(* CODESYS project Broadcast.library
   Company: _
   DefaultNamespace: Broadcast
   Title: Broadcast
   Placeholder: _Broadcast
   Author: Krystian Lis et al.
   Description: Sub-pub com.
   Version: 1.0.0

Project tree, tasks and I/O mapping:
  libraries: Debug, * (_); Results, * (_); Strings, * (_); Tags, * (_); Utils, * (_); Tc2_Standard, * (Beckhoff Automation GmbH); Tc2_System, * (Beckhoff Automation GmbH); Domains, * (_); Calls, * (_)
  Broadcast/
    _/
      Helpers/
        function _ArePaired [ST]
        function _Cleanup [ST]
        function _Clear [ST]
        function _Copy [ST]
        function _EmitSignal [ST]
        function _FindBestChunk [ST]
        function _FindChunkAfter [ST]
        function _NewPair [ST]
        function _SoftCompress [ST]
        function _Unpair [ST]
      Structs/
        data type ST_Entry
    Receiver/
      interface I_Receiver: Pair, Unpair
      interface I_ReceiverNode: IsOk, Receive
      function block Receiver [ST]: FB_init, IsOk, Pair, Receive, Tag, Unpair
    Signal/
      function block EmitProxy [ST]: FB_init
      interface I_Emit: Emit, EmitTo, Option, Pair, Unpair
      interface I_Signal: Pair, Unpair
      interface I_SignalNode: count, id, size
      function block Signal [ST]: count, id, size, Emit, EmitTo, FB_init, Option, Pair, Tag, Unpair
    global variables _Channel
    global variables Param
*)

// Broadcast/_/Structs/ST_Entry
TYPE INTERNAL ST_Entry :
STRUCT
	iSignal		: I_SignalNode;
	iReceiver	: I_ReceiverNode;
END_STRUCT
END_TYPE

// Broadcast/_Channel
{attribute 'qualified_only'}
VAR_GLOBAL INTERNAL
	{attribute 'ExpandFully'} 
	// Fixed-size array to store all signal-receiver entries.
	// Index 0 is reserved and not used (signals with id = 0 are unassigned).
	stEntry				: ARRAY[0..Param.nChannelSize] OF ST_Entry;
	
	// Total number of assigned entries in the stEntry array.
	nAssigned			: UDINT;
END_VAR

// Broadcast/Param
{attribute 'qualified_only'}
VAR_GLOBAL CONSTANT
	nChannelSize		: UDINT(1..16#FFFFFFE) := 100;
END_VAR

// Broadcast/_/Helpers/_ArePaired
FUNCTION INTERNAL _ArePaired : BOOL
VAR_INPUT
	iSignal				: I_SignalNode;
    iReceiver			: I_ReceiverNode;
END_VAR
VAR_OUTPUT
	nPos				: UDINT;
END_VAR
VAR
	i					: UDINT;
	_nEnd				: UDINT;
END_VAR

IF iSignal.count = 0 THEN
	_ArePaired := FALSE;
	RETURN;	
END_IF

_nEnd := iSignal.id + iSignal.count - 1;
FOR i := iSignal.id TO _nEnd DO
	IF _Channel.stEntry[i].iReceiver = iReceiver THEN
		_ArePaired := TRUE;
		nPos := i;
		RETURN;
	END_IF
END_FOR

END_FUNCTION

// Broadcast/Signal/I_SignalNode
INTERFACE INTERNAL I_SignalNode EXTENDS Debug.I_Debug

PROPERTY INTERNAL count : UDINT
GET
END_GET
SET
END_SET
END_PROPERTY

PROPERTY INTERNAL id : UDINT
GET
END_GET
SET
END_SET
END_PROPERTY

PROPERTY INTERNAL size : UDINT
GET
END_GET
SET
END_SET
END_PROPERTY

END_INTERFACE

// Broadcast/Receiver/I_ReceiverNode
INTERFACE INTERNAL I_ReceiverNode EXTENDS Debug.I_Debug

PROPERTY INTERNAL IsOk : BOOL
GET
END_GET
END_PROPERTY

METHOD INTERNAL Receive
VAR_INPUT
	iArg			: Calls.I_Arg;
END_VAR
END_METHOD

END_INTERFACE

// Broadcast/_/Helpers/_Cleanup
FUNCTION INTERNAL _Cleanup
VAR
	i					: UDINT;
	_iSignal			: I_SignalNode;
END_VAR

// Loop through stEntry to update signal ids
FOR i := 1 TO Param.nChannelSize DO
	IF _Channel.stEntry[i].iSignal <> 0 AND_THEN _Channel.stEntry[i].iSignal <> _iSignal THEN
			_iSignal := _Channel.stEntry[i].iSignal;
			_iSignal.id := i;
	END_IF
END_FOR

END_FUNCTION

// Broadcast/Signal/Signal
FUNCTION_BLOCK FINAL Signal IMPLEMENTS I_SignalNode, I_Signal, Tags.I_Tagged, I_Emit
VAR
	_tag			: Tags.Tag;
	_nCount			: UDINT;
	_nSize			: UDINT;
	_nId			: UDINT;
END_VAR

PROPERTY INTERNAL count : UDINT
GET
count := _nCount;
END_GET
SET
_nCount := count;
END_SET
END_PROPERTY

PROPERTY INTERNAL id : UDINT
GET
id := _nId;
END_GET
SET
_nId := id;
END_SET
END_PROPERTY

PROPERTY INTERNAL size : UDINT
GET
size := _nSize;
END_GET
SET
_nSize := size;
END_SET
END_PROPERTY

METHOD Emit
VAR_INPUT
	iArg			: Calls.I_Arg := 0;
END_VAR
IF iArg = 0 THEN
	iArg := Calls.Arg.phantom;
END_IF

_EmitSignal(THIS^, iArg);
END_METHOD

METHOD EmitTo : Results.Result
VAR_INPUT
	iReceiver		: I_Receiver;
	iArg			: Calls.I_Arg;
END_VAR
IF iReceiver = 0 THEN
	EmitTo := Results.Err.Itf0;
	RETURN;
END_IF

IF iArg = 0 THEN
	iArg := Calls.Arg.phantom;
END_IF

iReceiver.Receive(iArg);
EmitTo := Results.Ok;
END_METHOD

//FB_Init is always available implicitly and it is used primarily for initialization.
//The return value is not evaluated. For a specific influence, you can also declare the
//methods explicitly and provide additional code there with the standard initialization
//code. You can evaluate the return value.
METHOD FB_Init: BOOL
VAR_INPUT
    bInitRetains: BOOL; // TRUE: the retain variables are initialized (reset warm / reset cold)
    bInCopyCode: BOOL;  // TRUE: the instance will be copied to the copy code afterward (online change)

	iCTable		: Domains.I_MutCTable;
END_VAR
VAR
	_nResult		: Results.Result;
END_VAR
IF iCTable <> 0 THEN
	CASE (_nResult := iCTable.Insert(THIS^)) OF
		Results.Ok:	
			// Do nothing
		Results.Err.ItfEq:
			Debug.DebugMsg(THIS^, 'Alredy exist within iCTable!');
			Debug.DebugMsg(iCTable, '^');
		Results.Err.Ovf:
			Debug.DebugMsg(THIS^, 'iCTable overflow!');
		ELSE
			Debug.DebugMsg(THIS^, Tc2_Standard.CONCAT(TO_STRING(_nResult), ': Unknown error'));
	END_CASE

ELSE
	Debug.DebugMsg(THIS^, 'iCTable = 0!');
END_IF
END_METHOD

METHOD Option : REFERENCE TO Signal
VAR_INPUT
	sOption		: Strings.Str;
END_VAR
Option REF= THIS^;
_tag.Option := sOption;
END_METHOD

METHOD Pair : Results.Result
VAR_INPUT
	iReceiver		: I_Receiver;
END_VAR
IF iReceiver = 0 THEN
	Pair := Results.Err.Itf0;
ELSIF iReceiver.IsOk THEN
	Pair := _NewPair(THIS^, iReceiver);
ELSE
	Pair := Results.Error;
END_IF
END_METHOD

PROPERTY Tag : Tags.I_Tag
GET
Tag := _tag;
END_GET
END_PROPERTY

METHOD Unpair : Results.Result
VAR_INPUT
	iReceiver		: I_Receiver;
END_VAR
IF iReceiver = 0 THEN
	Unpair := Results.Err.Itf0;
ELSIF iReceiver.IsOk THEN
	Unpair := _Unpair(THIS^, iReceiver);
ELSE
	Unpair := Results.Error;
END_IF
END_METHOD

END_FUNCTION_BLOCK

// Broadcast/Signal/I_Signal
INTERFACE I_Signal EXTENDS Debug.I_Debug, Domains.I_Component

METHOD Pair : Results.Result
VAR_INPUT
	iReceiver		: I_Receiver;
END_VAR
END_METHOD

METHOD Unpair : Results.Result
VAR_INPUT
	iReceiver		: I_Receiver;
END_VAR
END_METHOD

END_INTERFACE

// Broadcast/Receiver/I_Receiver
INTERFACE I_Receiver EXTENDS I_ReceiverNode, Domains.I_Component;

METHOD Pair : Results.Result
VAR_INPUT
	iSignal		: I_Signal;
END_VAR
END_METHOD

METHOD Unpair : Results.Result
VAR_INPUT
	iSignal		: I_Signal;
END_VAR
END_METHOD

END_INTERFACE

// Broadcast/Signal/I_Emit
INTERFACE I_Emit

METHOD Emit
VAR_INPUT
	iArg			: Calls.I_Arg;
END_VAR
END_METHOD

METHOD EmitTo : Results.Result
VAR_INPUT
	iReceiver		: I_Receiver;
	iArg			: Calls.I_Arg;
END_VAR
END_METHOD

METHOD Option : REFERENCE TO Signal
VAR_INPUT
	sOption		: Strings.Str;
END_VAR
END_METHOD

METHOD Pair : Results.Result
VAR_INPUT
	iReceiver		: I_Receiver;
END_VAR
END_METHOD

METHOD Unpair : Results.Result
VAR_INPUT
	iReceiver		: I_Receiver;
END_VAR
END_METHOD

END_INTERFACE

// Broadcast/_/Helpers/_EmitSignal
FUNCTION INTERNAL _EmitSignal
VAR_INPUT
	iSignal		: I_SignalNode;
	iArg		: Calls.I_Arg;
END_VAR
VAR
	i			: UDINT;
	nEnd		: UDINT;
END_VAR

IF iSignal.count = 0 THEN
	RETURN;
END_IF

nEnd := iSignal.id + iSignal.count - 1;
FOR i := iSignal.id TO nEnd DO
	_Channel.stEntry[i].iReceiver.Receive(iArg);
END_FOR

END_FUNCTION

// Broadcast/_/Helpers/_NewPair
FUNCTION INTERNAL _NewPair : Results.Result
VAR_INPUT
	iSignal				: I_SignalNode;
	iReceiver			: I_ReceiverNode;
END_VAR
VAR
	_nSignalSize		: UDINT;
	_nSignalCount		: UDINT;
	_nSignalId			: UDINT;
	
	_nNewId				: UDINT;
	_nNewSize			: UDINT;
	_nRequestedSize		: UDINT;
	_nDiff				: UDINT;
	
	_nFree				: UDINT;
	
	_bReallocation		: BOOL;
END_VAR

//If itfs are 0
IF iSignal = 0 OR iReceiver = 0 THEN
	_NewPair := Results.Err.Itf0;
	RETURN;
END_IF	
//If pair already exist
IF _ArePaired(iSignal, iReceiver) THEN
	_NewPair := Results.None;
	RETURN;
END_IF
// First signal ever
IF _Channel.nAssigned = 0 THEN
	_Channel.stEntry[1].iSignal := iSignal;
	_Channel.stEntry[1].iReceiver := iReceiver;
	iSignal.id := 1;
	iSignal.size := 1;
	iSignal.count := 1;
	_Channel.nAssigned := 1;;
	_NewPair := Results.Ok;
	RETURN;	
END_IF

//If signal has enough space
IF (_nSignalCount := iSignal.count) > 0 AND_THEN _nSignalCount < (_nSignalSize := iSignal.size) THEN
	_Channel.stEntry[iSignal.id + _nSignalCount].iSignal := iSignal;
	_Channel.stEntry[iSignal.id + _nSignalCount].iReceiver := iReceiver;
	iSignal.count := _nSignalCount + 1;
	_NewPair := Results.Ok;
	RETURN;
END_IF

IF iSignal.id <> 0 THEN
	//If signal has enough space after
	IF Results.IsOk(_FindChunkAfter(_nSignalSize + (_nSignalId := iSignal.id), 1, nNewSize => _nNewSize)) THEN
		_Channel.stEntry[iSignal.id + _nSignalCount].iSignal := iSignal;
		_Channel.stEntry[iSignal.id + _nSignalCount].iReceiver := iReceiver;
		iSignal.size := _nNewSize + _nSignalSize;
		iSignal.count := _nSignalCount + 1;
		_Channel.nAssigned := _Channel.nAssigned + 1;
		_NewPair := Results.Ok;
		RETURN;
	END_IF
END_IF

// What new size should be
IF (_nFree := Param.nChannelSize - _Channel.nAssigned) >= _nSignalSize + 1 THEN
	_nRequestedSize := _nSignalSize + 1;
ELSE
	_NewPair := Results.Err.Ovf;
	RETURN;
END_IF

_nSignalId := iSignal.id;
IF Results.IsOk(_FindBestChunk(_nSignalId, _nRequestedSize, nNewId => _nNewId, nNewSize => _nNewSize)) THEN
	IF _nSignalId <> 0 THEN
		_Copy(_nSignalId, _nSignalSize, _nNewId);
		_Clear(_nSignalId, _nSignalSize);		
	END_IF		
	_Channel.stEntry[_nNewId + _nSignalCount].iSignal := iSignal;
	_Channel.stEntry[_nNewId + _nSignalCount].iReceiver := iReceiver;
	iSignal.id := _nNewId;
	iSignal.size := _nNewSize;
	iSignal.count := _nSignalCount + 1;
	_Channel.nAssigned := _Channel.nAssigned - _nSignalSize + _nNewSize;
	_NewPair := Results.Ok;	
	RETURN;
END_IF

_SoftCompress();
_Cleanup();


_nSignalId := iSignal.id; // _nSignalId needs to be revalidated.
IF Results.IsOk(_FindBestChunk(_nSignalId, _nRequestedSize, nNewId => _nNewId, nNewSize => _nNewSize)) THEN
	IF _nSignalId <> 0 THEN
		_Copy(_nSignalId, _nSignalSize, _nNewId);
		_Clear(_nSignalId, _nSignalSize);		
	END_IF
	_Channel.stEntry[_nNewId + _nSignalCount].iSignal := iSignal;
	_Channel.stEntry[_nNewId + _nSignalCount].iReceiver := iReceiver;
	iSignal.id := _nNewId;
	iSignal.size := _nNewSize;
	iSignal.count := _nSignalCount + 1;
	_Channel.nAssigned := _Channel.nAssigned - _nSignalSize + _nNewSize;
	_NewPair := Results.Ok;	
	RETURN;
END_IF

_NewPair := Results.Error;

END_FUNCTION

// Broadcast/_/Helpers/_FindChunkAfter
FUNCTION INTERNAL _FindChunkAfter : Results.Result
VAR_INPUT
	nId					: UDINT;
    nRequestedSize     	: UDINT;
END_VAR
VAR_OUTPUT
    nNewSize            : UDINT;
END_VAR
VAR
	i					: UDINT;
END_VAR

// Loop from the starting index to the end of stEntry
FOR i := nId TO Param.nChannelSize DO
	IF nRequestedSize = nNewSize THEN
		EXIT;
	ELSIF _Channel.stEntry[i].iSignal = 0 THEN
		nNewSize := nNewSize + 1;
	ELSE
		EXIT;
	END_IF
END_FOR

// Check if the required size was found
IF nNewSize = nRequestedSize THEN
	_FindChunkAfter := Results.Ok;
ELSE
	_FindChunkAfter := Results.Error;
END_IF

END_FUNCTION

// Broadcast/_/Helpers/_FindBestChunk
FUNCTION INTERNAL _FindBestChunk : Results.Result
VAR_INPUT
	nRequesterId		: UDINT;
    nRequestedSize     	: UDINT;
END_VAR
VAR_OUTPUT
    nNewId             	: UDINT;
    nNewSize            : UDINT;
END_VAR
VAR
	i					: UDINT;
	j					: UDINT;
END_VAR

// Loop through stEntry to find the best chunk
FOR i := 1 TO Param.nChannelSize DO
	IF _Channel.stEntry[i].iSignal <> 0 AND_THEN _Channel.stEntry[i].iSignal.id <> nRequesterId THEN
		// Skip over occupied blocks
		i := _Channel.stEntry[i].iSignal.id + _Channel.stEntry[i].iSignal.size - 1;
	ELSE
		// Start of a free chunk and measure its size
		FOR j := 0 TO Param.nChannelSize DO
			IF _Channel.stEntry[i + j].iSignal <> 0 AND_THEN _Channel.stEntry[i].iSignal.id <> nRequesterId THEN
				EXIT;
			ELSIF Param.nChannelSize <= i + j THEN
				EXIT;
			END_IF			
		END_FOR
		
		// If the chunk is smaller but still fits assign a new best fit
		IF nNewSize = 0 THEN
			nNewId := i;
			nNewSize := j + 1;
		ELSIF  nRequestedSize <= j + 1 AND_THEN nNewSize > j + 1 THEN
			nNewId := i;
			nNewSize := nRequestedSize;
		END_IF
		
		IF _Channel.stEntry[i + j].iSignal = 0 THEN
			i := i + j;
		ELSE
			i := i + j - 1;
		END_IF
		
	END_IF
END_FOR

IF nNewSize > 0 THEN
	nNewSize := nRequestedSize;
	_FindBestChunk := Results.Ok;
ELSE
	_FindBestChunk := Results.Error;
END_IF

END_FUNCTION

// Broadcast/_/Helpers/_Copy
FUNCTION INTERNAL _Copy : Results.Result;
VAR_INPUT
	nOldId		: UDINT;
	nOldSize	: UDINT;
	nNewId		: UDINT;
END_VAR

IF Results.IsNone(UDINT_TO_INT(Tc2_System.MEMMOVE(ADR(_Channel.stEntry[nNewId]), ADR(_Channel.stEntry[nOldId]), nOldSize * SIZEOF(ST_Entry)))) THEN
	_Copy := Results.Err.TcLib;
ELSE
	_Copy := Results.Ok;
END_IF

END_FUNCTION

// Broadcast/_/Helpers/_Clear
FUNCTION INTERNAL _Clear : Results.Result
VAR_INPUT
	nId		: UDINT;
	nSize	: UDINT;
END_VAR

IF Results.IsNone(UDINT_TO_INT(Tc2_SYSTEM.MEMSET(ADR(_Channel.stEntry[nId]), 0, SIZEOF(ST_Entry) * nSize))) THEN
	_Clear := Results.Err.TcLib;
ELSE
	_Clear := Results.Ok;
END_IF

END_FUNCTION

// Broadcast/_/Helpers/_SoftCompress
FUNCTION INTERNAL _SoftCompress
VAR
	i			: UDINT;
	_nFreePtr	: UDINT;
	_stEmpty	: ST_Entry;	
END_VAR

// Find the first free entry in stEntry
FOR i := 1 TO Param.nChannelSize DO
	IF _Channel.stEntry[i].iSignal <> 0 THEN
		i := _Channel.stEntry[i].iSignal.id + _Channel.stEntry[i].iSignal.size - 1;
	ELSE
		_nFreePtr := i;
	END_IF
END_FOR

// If no free entry found, no need to compress
IF _nFreePtr = 0 THEN
	RETURN;
END_IF 

// Move entries to fill the free space
FOR i := _nFreePtr TO Param.nChannelSize DO
	IF _Channel.stEntry[i].iSignal <> 0 AND_THEN _nFreePtr > 0 THEN
		_Channel.stEntry[_nFreePtr] := _Channel.stEntry[i];
		_Channel.stEntry[i] := _stEmpty;
	ELSE
		_nFreePtr := i;
	END_IF
END_FOR

END_FUNCTION

// Broadcast/_/Helpers/_Unpair
FUNCTION INTERNAL _Unpair : Results.Result
VAR_INPUT
	iSignal		: I_SignalNode;
	iReceiver	: I_ReceiverNode;
END_VAR
VAR
	i			: UDINT;
	_nPos		: UDINT;
	_nEnd		: UDINT;
	_nCount		: UDINT;
END_VAR

IF iSignal = 0 OR iReceiver = 0 THEN
	_Unpair := Results.Err.Itf0;
	RETURN;
END_IF

IF NOT _ArePaired(iSignal, iReceiver, nPos => _nPos) THEN
	_Unpair := Results.None;
	RETURN;
END_IF

_nCount := iSignal.count;
_nEnd := iSignal.id + _nCount - 1;

// Swap with the last receiver if not already the last
IF _nPos <> _nEnd THEN
	_Channel.stEntry[_nPos] := _Channel.stEntry[_nEnd];
END_IF

// Clear the last entry
_Channel.stEntry[_nEnd].iSignal := 0;
_Channel.stEntry[_nEnd].iReceiver := 0;

// Update counts
iSignal.count := _nCount - 1;
_Channel.nAssigned := _Channel.nAssigned - 1;

// Shrink if needed
IF iSignal.count < iSignal.size / 2 THEN
	iSignal.size := iSignal.count;
END_IF

_Unpair := Results.Ok;

END_FUNCTION

// Broadcast/Receiver/Receiver
FUNCTION_BLOCK FINAL Receiver IMPLEMENTS I_ReceiverNode, I_Receiver, Tags.I_Tagged
VAR
	_iReceiver		: Calls.I_Call;
	_tag			: Tags.Tag;
	_bIsOk			: BOOL := TRUE;
END_VAR

//FB_Init is always available implicitly and it is used primarily for initialization.
//The return value is not evaluated. For a specific influence, you can also declare the
//methods explicitly and provide additional code there with the standard initialization
//code. You can evaluate the return value.
METHOD FB_Init: BOOL
VAR_INPUT
    bInitRetains: BOOL; // TRUE: the retain variables are initialized (reset warm / reset cold)
    bInCopyCode: BOOL;  // TRUE: the instance will be copied to the copy code afterward (online change)

	iCTable		: Domains.I_MutCTable;
	iReceiver	: Calls.I_Call;
END_VAR
VAR
	_nResult	: Results.Result;
END_VAR
_iReceiver := iReceiver;
IF _iReceiver = 0 THEN
	_bIsOk := FALSE;
	Debug.DebugMsg(THIS^, 'iReceiver = 0!');
END_IF

IF iCTable = 0 THEN
	_bIsOk := FALSE;
	Debug.DebugMsg(THIS^, 'iCTable = 0!');
END_IF

IF NOT _bIsOk THEN
	RETURN;
END_IF

CASE (_nResult := iCTable.Insert(THIS^)) OF
	Results.Ok:	
		// Do nothing
	Results.Err.ItfEq:
		Debug.DebugMsg(THIS^, 'Alredy exist within iCTable!');
		Debug.DebugMsg(iCTable, '^');
		_bIsOk := FALSE;
	Results.Err.Ovf:
		Debug.DebugMsg(THIS^, 'iCTable overflow!');
		_bIsOk := FALSE;
	ELSE
		Debug.DebugMsg(THIS^, Tc2_Standard.CONCAT(TO_STRING(_nResult), ': Unknown error!'));
		_bIsOk := FALSE;
END_CASE
END_METHOD

PROPERTY INTERNAL IsOk : BOOL
GET
IsOk := _bIsOk;
END_GET
END_PROPERTY

METHOD Pair : Results.Result
VAR_INPUT
	iSignal		: I_Signal;
END_VAR
IF iSignal <> 0 THEN
	Pair := iSignal.Pair(THIS^);
ELSE
	Pair := Results.Error;
END_IF
END_METHOD

METHOD INTERNAL Receive
VAR_INPUT
	iArg			: Calls.I_Arg;
END_VAR
_iReceiver.Call(iArg);
END_METHOD

PROPERTY Tag : Tags.I_Tag
GET
Tag := _tag;
END_GET
END_PROPERTY

METHOD Unpair : Results.Result
VAR_INPUT
	iSignal		: I_Signal;
END_VAR
IF iSignal <> 0 THEN
	Unpair := iSignal.Unpair(THIS^);
ELSE
	Unpair := Results.Error;
END_IF
END_METHOD

END_FUNCTION_BLOCK

// Broadcast/Signal/EmitProxy
FUNCTION_BLOCK EmitProxy IMPLEMENTS Debug.I_Debug
VAR_INPUT
END_VAR
VAR_OUTPUT
END_VAR
VAR
END_VAR

//FB_Init is always available implicitly and it is used primarily for initialization.
//The return value is not evaluated. For a specific influence, you can also declare the
//methods explicitly and provide additional code there with the standard initialization
//code. You can evaluate the return value.
METHOD FB_Init: BOOL
VAR_INPUT
    bInitRetains: BOOL; // TRUE: the retain variables are initialized (reset warm / reset cold)
    bInCopyCode: BOOL;  // TRUE: the instance will be copied to the copy code afterward (online change)
	
	iEmit			: I_Emit;
	refEmitProxy	: REFERENCE TO I_Emit;	
	
END_VAR
IF iEmit = 0 THEN
	Debug.DebugMsg(THIS^, 'iEmit = 0!');
	RETURN;
END_IF

IF __ISVALIDREF(refEmitProxy) THEN
	refEmitProxy := iEmit;
ELSE
	Debug.DebugMsg(THIS^, 'refEmitProxy ref invalid!');
END_IF
END_METHOD

END_FUNCTION_BLOCK
